PROGRAM P_List_Example
VAR
	fbList 		: FB_List;
	sData 		: STRING;
	sRTNData	: ARRAY[0..3] OF STRING;
	nCount 		: DINT;
	eState 		: (CREATE, REVERSE, REMOVE, COUNT, IDLE);
	stError 	: ST_ERROR;
END_VAR

stError := fbList._Error_Status;// (stError => stError);
CASE eState OF
	CREATE:
		sData := 'Cats';fbList.Create(sData);
		sData := 'Dogs';fbList.Create(sData);
		sData := 'Birds';fbList.Create(sData);
		sData := 'Fish';fbList.Insert(sData, 1);

		fbList.Get(sRTNData[0], 0)
			  .Get(sRTNData[1], 1)
			  .Get(sRTNData[2], 2)
			  .Get(sRTNData[3], 3);
		eState := IDLE;
	REVERSE:
		fbList.Reverse();
		fbList.Get(sRTNData[0], 0)
			  .Get(sRTNData[1], 1)
			  .Get(sRTNData[2], 2)
			  .Get(sRTNData[3], 3);
		eState := IDLE;
	REMOVE:
		fbList.RemoveAt(2)
			  .Get(sRTNData[0], 0)
			  .Get(sRTNData[1], 1)
			  .Get(sRTNData[2], 2)
			  .Get(sRTNData[3], 3);
		eState := IDLE;
	COUNT: 
		nCount := fbList._Count;
		eState := IDLE;
		
		
END_CASE

END_PROGRAM

(* stored: Version 1.1.0.1, ProductVersion 3.1.4024.4
   POU P_List_Example: Id {a33a4cf6-5cec-400c-8295-07b960a43c21}, SpecialFunc None *)
